(* PLC project Rasi_feeds_batching2.project, Automation Builder 2.7 - Basic Automation Builder 2.7 *)
(* stored: creationDateTime 2026-09-01T00:26:23.0508492, modificationDateTime 2026-09-01T00:24:44.1606357 *)

FUNCTION_BLOCK sample_read_two_weights
  VAR_INPUT
    Enable : BOOL := TRUE;
    Com_Slot : BYTE := 1;
    Slave_Auto_ID : BYTE := 1;
    Slave_Semi_ID : BYTE := 2;
    iDivisor_Auto : REAL := 10.0;
    iDivisor_Semi : REAL := 10.0;
    Tare_Auto : BOOL;
    Tare_Semi : BOOL;
  END_VAR
  VAR_OUTPUT
    Weight_Auto : REAL;
    Weight_Semi : REAL;
    Auto_Fault : BOOL;
    Semi_Fault : BOOL;
    Bus_Busy : BOOL;
    Active_Node : BYTE;
  END_VAR
  VAR
    fbMulti : FB_Samyak_Multi;
    arrSlaves : ARRAY[1..4] OF BYTE := [1, 2, 0, 0];
    arrDiv : ARRAY[1..4] OF REAL := [10.0, 10.0, 1.0, 1.0];
    arrTare : ARRAY[1..4] OF BOOL;
    Weight_Scaled_Array : ARRAY[1..4] OF REAL;
    Line_Fault_Array : ARRAY[1..4] OF BOOL;
  END_VAR

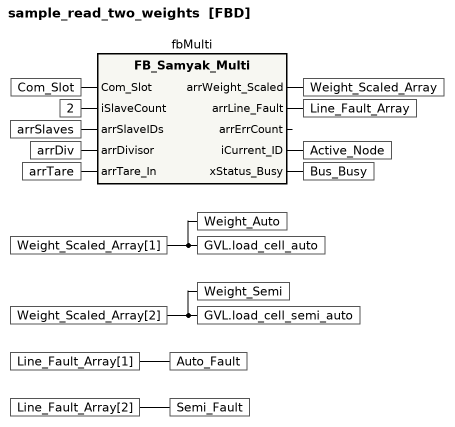
(* FBD diagram, written out as Structured Text *)
fbMulti(Com_Slot := Com_Slot, iSlaveCount := 2, arrSlaveIDs := arrSlaves, arrDivisor := arrDiv, arrTare_In := arrTare, arrLine_Fault => Line_Fault_Array, iCurrent_ID => Active_Node, xStatus_Busy => Bus_Busy);
Weight_Scaled_Array := fbMulti.arrWeight_Scaled;
Weight_Auto := Weight_Scaled_Array[1];
GVL.load_cell_auto := Weight_Scaled_Array[1];
Weight_Semi := Weight_Scaled_Array[2];
GVL.load_cell_semi_auto := Weight_Scaled_Array[2];
Auto_Fault := Line_Fault_Array[1];
Semi_Fault := Line_Fault_Array[2];
END_FUNCTION_BLOCK
